PROGRAM main
  VAR
    HS101A_PBGreen AT %IX0.0 : BOOL; (* Green push button *)
    HS101B_PBYellow AT %IX0.1 : BOOL; (* Yellow push button *)
    HS101C_PBRed AT %IX0.2 : BOOL; (* Red push button *)
    XL101A_Green AT %QX0.0 : BOOL; (* Green light *)
    XL101B_Yellow AT %QX0.1 : BOOL; (* Yellow light *)
    XL101C_Red AT %QX0.2 : BOOL; (* Red light *)
  END_VAR

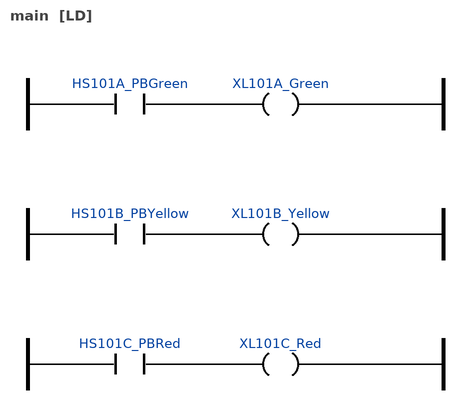
(* LD diagram, written out as Structured Text *)
XL101A_Green := HS101A_PBGreen;
XL101B_Yellow := HS101B_PBYellow;
XL101C_Red := HS101C_PBRed;
END_PROGRAM
